PROGRAM START_STOP_1
VAR
	START_TIMER : TON;
	START_TIMER_ELAPSED: TIME;
	START_TIMER_DONE : BOOL; 
	START_PB AT %I*:BOOL;
	STOP_PB AT %I*:BOOL;
	START_REQUEST:BOOL;
	STOP_REQUEST:BOOL;


END_VAR
VAR // added by the converter: edge detectors and wires of the graphical bodies
    _rt1 : R_TRIG;
END_VAR

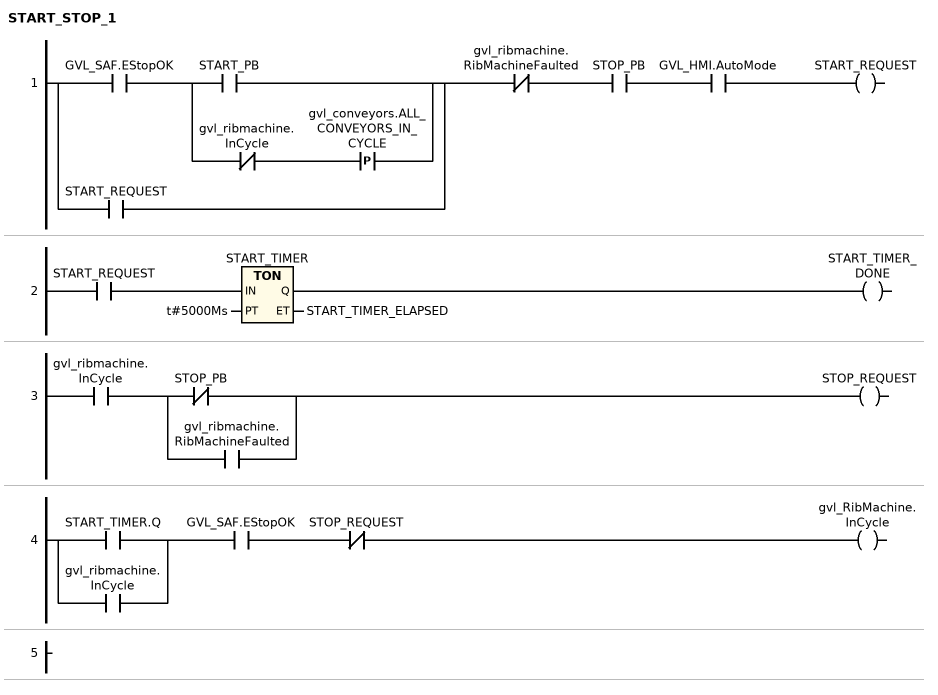
// NETWORK 1
_rt1(CLK := gvl_conveyors.ALL_CONVEYORS_IN_CYCLE);
START_REQUEST := (GVL_SAF.EStopOK AND (START_PB OR NOT gvl_ribmachine.InCycle AND _rt1.Q) OR START_REQUEST) AND NOT gvl_ribmachine.RibMachineFaulted AND STOP_PB AND GVL_HMI.AutoMode;

// NETWORK 2
START_TIMER(IN := START_REQUEST, PT := t#5000Ms, ET => START_TIMER_ELAPSED); // TON
START_TIMER_DONE := START_TIMER.Q;

// NETWORK 3
STOP_REQUEST := gvl_ribmachine.InCycle AND (NOT STOP_PB OR gvl_ribmachine.RibMachineFaulted);

// NETWORK 4
gvl_RibMachine.InCycle := (START_TIMER.Q OR gvl_ribmachine.InCycle) AND GVL_SAF.EStopOK AND NOT STOP_REQUEST;

// NETWORK 5

END_PROGRAM

(* stored: Version 1.1.0.1, ProductVersion 3.1.4024.12
   POU START_STOP_1: Id {ad44f4f2-2216-4aa1-a9da-467f8b8e19f2}, SpecialFunc None *)
